TYPE
	tchmi_framework_definitions_XtsMoverListItem :
	STRUCT
		MoverIndex          : UINT (* minimum value: 0 maximum value: 65535 *) ;
		ProcessingUnitIndex : UINT (* minimum value: 0 maximum value: 65535 *) ;
	END_STRUCT
END_TYPE

(* stored: Version 1.1.0.1, ProductVersion 3.1.4024.12
   DUT tchmi_framework_definitions_XtsMoverListItem: Id {a0b8e178-c6ab-4614-8df4-efe9468eeb61} *)
